// TIA Portal V18 export
DATA_BLOCK "HomePosManagerDb"   // DB65
VERSION : 0.1
// stored: AutoNumber true, DBAccessibleFromOPCUA true, InstanceOfName _hmi_singleSpotManager, InstanceOfType FB
"_hmi_singleSpotManager"
   // VAR_INPUT
   //    hmi_PosSet : "typePositions";
   //    cur_pos_set : "typePositions";
   // END_VAR
   // VAR_IN_OUT
   //    hmiFromHmi : Bool;
   //    hmiSFromEncoder : Bool;
   //    posToModify : "typePositions";
   // END_VAR
   // VAR
   //    N_max : Int;
   // END_VAR
BEGIN
END_DATA_BLOCK
